Universal Robots PolyScope program: reciprocal_p2_2.urp

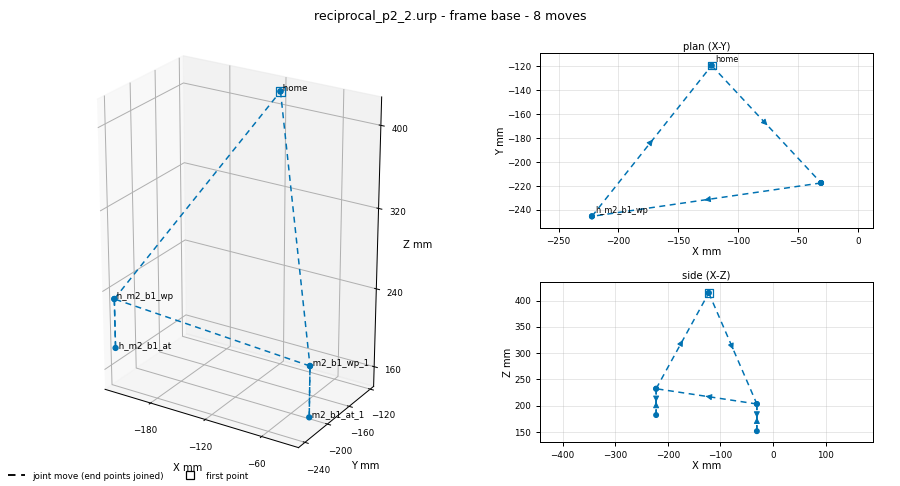
[picture p0: tool path of reciprocal_p2_2.urp in frame base, 8 of 8 moves have a stored position in this frame; points joined in program order, loops and branches not executed]
Program reciprocal_p2_2 (installation=default_1 directory=/programs/../media/urmountpoint_GSJLiG/ITER createdIn=5.3.1.64192 lastSavedIn=5.3.1.64192 robotSerialNumber=20195300365)
Calibrated DH parameters: a=[-0.000093, -0.190649, -0.212673, 0.000091, -0.000205, 0]; d=[0.151591, 44.061648, -42.488068, -1.442789, 0.085322, 0.091911]; alpha=[1.570082, -0.003447, 0.007513, 1.572293, -1.571904, 0]; deltaTheta=[0, -0.672656, 0.728185, -0.055522, 0.000005, 0]
Robot Program (runOnlyOnce=false)
  URCap Gripper Activate (Robotiq_Grippers, Robotiq Inc.) dataModel(ResetAndActivateKey=false)
  URCap Gripper (Robotiq_Grippers, Robotiq Inc.) dataModel(position=50.0, force=100.0, speed=100.0, positionInDouble=50.0, forceInDouble=100.0, speedInDouble=100.0, slaveIds=[9], blocking=true)
  MoveJ speed 60 deg/s, acceleration 80 deg/s^2 (useActiveTCP=true) feature=Base
    Waypoint home: TCP in base x=-122.15 y=-119.32 z=414.454 mm, rx=2.2563 ry=2.1459 rz=-0.0481 rad; joints [-85.681, -56.776, -79.802, -131.025, 89.944, -262.833] deg
  Folder Mid_2
    MoveJ speed 60 deg/s, acceleration 80 deg/s^2 (useActiveTCP=true) feature=Base
      Waypoint m2_b1_wp_1: TCP in base x=-30.704 y=-217.422 z=203.363 mm, rx=-2.2397 ry=-2.1922 rz=0.0003 rad; joints [-61.845, -63.917, -136.913, -69.519, 90.279, -240.21] deg
      Waypoint m2_b1_at_1: TCP in base x=-30.716 y=-217.427 z=151.677 mm, rx=-2.2397 ry=-2.1922 rz=0.0003 rad; joints [-61.887, -74.21, -147.891, -48.249, 90.169, -240.122] deg
      URCap Gripper (Robotiq_Grippers, Robotiq Inc.) dataModel(position=100.0, force=100.0, speed=100.0, positionInDouble=100.0, forceInDouble=100.0, speedInDouble=100.0, slaveIds=[9], blocking=true)
      Waypoint m2_b1_wp_2: TCP in base x=-30.704 y=-217.422 z=203.363 mm, rx=-2.2397 ry=-2.1922 rz=0.0003 rad; joints [-61.845, -63.917, -136.913, -69.519, 90.279, -240.21] deg
      Waypoint h_m2_b1_wp: TCP in base x=-222.193 y=-245.34 z=232.403 mm, rx=-3.1314 ry=0.0205 rz=0.0123 rad; joints [-108.936, -94.247, -105.13, -70.966, 89.712, -197.837] deg
      Waypoint h_m2_b1_at: TCP in base x=-222.194 y=-245.343 z=182.32 mm, rx=-3.1314 ry=0.0205 rz=0.0122 rad; joints [-108.96, -99.771, -113.792, -56.782, 89.658, -197.776] deg
      URCap Gripper (Robotiq_Grippers, Robotiq Inc.) dataModel(position=50.0, force=100.0, speed=100.0, positionInDouble=50.0, forceInDouble=100.0, speedInDouble=100.0, slaveIds=[9], blocking=true)
      Waypoint h_m2_b1_wp: TCP in base x=-222.193 y=-245.34 z=232.403 mm, rx=-3.1314 ry=0.0205 rz=0.0123 rad; joints [-108.936, -94.247, -105.13, -70.966, 89.712, -197.837] deg
  MoveJ speed 60 deg/s, acceleration 80 deg/s^2 (useActiveTCP=true) feature=Base
    Waypoint home: TCP in base x=-122.15 y=-119.32 z=414.454 mm, rx=2.2563 ry=2.1459 rz=-0.0481 rad; joints [-85.681, -56.776, -79.802, -131.025, 89.944, -262.833] deg
